TYPE T_Ctrl_SIf_MTR_Cfg :
STRUCT
END_STRUCT
END_TYPE

(* stored: Version 1.1.0.1, ProductVersion 3.1.0.23
   DUT T_Ctrl_SIf_MTR_Cfg: Id {129e4afd-fa92-4ce2-96bd-8ddc654c9a3c} *)
